(* CoDeSys 2.3 export: ST_PumpDiagnostics.exp *)

(* Data type in Pump *)
(* ґШРУЭЮбвШЪР ЭРбЮбР *)
TYPE ST_PumpDiagnostics :
STRUCT
    (* ДЫРУШ бЮбвЮпЭШп *)
    xDryRun : BOOL;                (* БгеЮЩ еЮФ *)
    xClosedValve : BOOL;           (* ·РЪалвРп ЧРФТШЦЪР *)
    xCavitation : BOOL;            (* єРТШвРжШп *)
    xOverload : BOOL;              (* їХаХУагЧЪР *)
    xLowFlow : BOOL;              (* ЅШЧЪШЩ аРбеЮФ *)
    xHighFlow : BOOL;             (* ІлбЮЪШЩ аРбеЮФ *)
    xLowInletPressure : BOOL;     (* ЅШЧЪЮХ ФРТЫХЭШХ ЭР ТеЮФХ *)
    xHighOutletPressure : BOOL;   (* ІлбЮЪЮХ ФРТЫХЭШХ ЭР ТлеЮФХ *)
    xLowEfficiency : BOOL;        (* ЅШЧЪШЩ єїґ *)
    xMechanicalWear : BOOL;       (* јХеРЭШзХбЪШЩ ШЧЭЮб *)
    
    (* БзХвзШЪШ Ш ЭРаРСЮвЪР *)
    dwRunningHours : DWORD;        (* ЅРаРСЮвЪР, зРбл *)
    dwStartCount : DWORD;          (* єЮЫШзХбвТЮ ЯгбЪЮТ *)
    
    (* ВаХЭФл *)
    rAvgEfficiency : REAL;         (* БаХФЭШЩ єїґ *)
    rAvgPower : REAL;              (* БаХФЭпп ЬЮйЭЮбвм *)
    rTotalVolume : REAL;           (* ѕСйШЩ ЮСкХЬ ЯХаХЪРзЪШ *)
    
    (* єЮФл ФШРУЭЮбвШЪШ *)
    wDiagnosticCode : WORD;        (* єЮФ ФШРУЭЮбвШЪШ *)
    sDiagnosticMessage : STRING(80); (* БЮЮСйХЭШХ ФШРУЭЮбвШЪШ *)
END_STRUCT
END_TYPE
